// TIA Portal V17 export
// export: Created 2023-09-14T22:30:54.9161637Z, ExportSetting WithDefaults, DisplayName Totally Integrated Automation Portal, DisplayVersion V17 Update 6, DisplayName TIA Portal Openness, DisplayVersion V17 Update 6, DisplayName TIA Portal Teamcenter Gateway, DisplayVersion V17 Update 6, DisplayName TIA Portal Version Control Interface, DisplayVersion V17, DisplayName Simotion SCOUT TIA, DisplayVersion 5.4.3.0, DisplayName TIA Portal Test Suite Advanced, DisplayVersion V17 Update 1, DisplayName SIMOCODE ES, DisplayVersion V17 Update 5, DisplayName SINAMICS Startdrive Advanced, DisplayVersion V17 SP1, DisplayName SINAMICS Startdrive G130, G150, S120, S150, SINAMICS MV, S210, DisplayVersion V17 SP1, DisplayName SINAMICS Startdrive G110M, G120, G120C, G120D, G120P, G115D, DisplayVersion V17 SP1, DisplayName SIRIUS Safety ES, DisplayVersion V17 Update 5, DisplayName STEP 7 Professional, DisplayVersion V17 Update 6, DisplayName STEP 7 CFC, DisplayVersion V17 Update 1, DisplayName STEP 7 Safety, DisplayVersion V17 Update 6, DisplayName WinCC Advanced, DisplayVersion V17 Update 6, DisplayName SIMATIC Visualization Architect, DisplayVersion V17 Update 5
DATA_BLOCK "08_AL_FILTER"   // DB26
{ S7_Optimized_Access := 'TRUE' }
VERSION : 0.1
// stored: AutoNumber true, DBAccessibleFromOPCUA true, DBAccessibleFromWebserver true, IsOnlyStoredInLoadMemory false, IsRetainMemResEnabled false, IsWriteProtectedInAS false, MemoryReserve 100
   VAR
      "n0006-zp001-el001-k25501_SN50" : Bool;
      "n0007-zp001-el001-k25502_SN50" : Bool;
      "n0008-zp001-el001-k25601_SN50" : Bool;
      "n0009-zp001-el001-k25602_SN50" : Bool;
      "n0005-zp001-el001-k40001_SN50" : Bool;
      "n0013-uf317-xn10_SN50" : Bool;
      "n0015-uc16-el001-k30001_SN50" : Bool;
      "n0016-uc164-xn10_SN50" : Bool;
      "n0017-lv004-el001-k30001_SN50" : Bool;
      "n0018-lv004-el001-k30001_SN50" : Bool;
      "n0020-uc15-el001-k30001_SN50" : Bool;
      "n0023-uc154-xn10_SN50" : Bool;
      "n0021-icg11-el001-k30001_SN50" : Bool;
      "n0022-icg21-el001-k30001_SN50" : Bool;
      "n0025-uc14-el001-k30001_SN50" : Bool;
      "n0026-uc144-xn10_SN50" : Bool;
      "n0038-uc1-el001-k30001_SN50" : Bool;
      "n0039-lv001-el001-k30001_SN50" : Bool;
      "n0040-lv001-el001-k30001_SN50" : Bool;
      "n0041-uf31-el002-k30001_SN50" : Bool;
      "n0042-uf41-el002-k30001_SN50" : Bool;
      "n0044-ct1-el001-k30001_SN50" : Bool;
      "n0045-ct1-el002-k30001_SN50" : Bool;
      "n0046-ct1-el003-k30001_SN50" : Bool;
      "n0047-lv002-el001-k30001_SN50" : Bool;
      "n0048-lv002-el001-k30001_SN50" : Bool;
      "n0050-uc13-el001-k30001_SN50" : Bool;
      "n0051-uc134-xn10_SN50" : Bool;
      "n0053-uc12-el001-k30001_SN50" : Bool;
      "n0055-uc124-xn10_SN50" : Bool;
      "n0054-uf31-el003-k30001_SN50" : Bool;
      "n0057-uc11-el001-k30001_SN50" : Bool;
      "n0060-uc114-xn10_SN50" : Bool;
      "n0058-lv003-el001-k30001_SN50" : Bool;
      "n0059-lv003-el001-k30001_SN50" : Bool;
      "n0028-uc17-el001-k30001_SN50" : Bool;
      "n0029-uc173-xn10_SN50" : Bool;
      "n0010-zp001-el001-k24501_SN50" : Bool;
      "n0033-zp001-el001-k40001_SN50" : Bool;
      "n0034-ug6-el001-k30001_SN50" : Bool;
      "n0035-ug6-xn10_SN50" : Bool;
      "n0043-db93-el001-k30001_SN50" : Bool;
      "n0031-db931-xn10_SN50" : Bool;
      "n0005-lv008-el001-k30001_SN51" : Bool;
      "n0006-lv008-el001-k30001_SN51" : Bool;
      "n0007-icg22-el001-k30001_SN51" : Bool;
      "n0008-icg12-el001-k30001_SN51" : Bool;
      "n0009-uf42-el002-k30001_SN51" : Bool;
      "n0010-lv007-el001-k30001_SN51" : Bool;
      "n0011-lv007-el001-k30001_SN51" : Bool;
      "n0021-uc2-el001-k30001_SN51" : Bool;
      "n0025-dc91-el001-k30001_SN51" : Bool;
      "n0026-uc915-xn10_SN51" : Bool;
      "n0027-uc915-xn11_SN51" : Bool;
      "n0028-lv005-el001-k30001_SN51" : Bool;
      "n0029-ct2-el001-k30001_SN51" : Bool;
      "n0033-uc26-el001-k30001_SN51" : Bool;
      "n0034-uc264-xn10_SN51" : Bool;
      "n0035-ct2-el002-k30001_SN51" : Bool;
      "n0036-lv005-el001-k30001_SN51" : Bool;
      "n0041-uc27-el001-k30001_SN51" : Bool;
      "n0042-uc274-xn10_SN51" : Bool;
      "n0046-uc25-el001-k30001_SN51" : Bool;
      "n0047-uc254-xn10_SN51" : Bool;
      "n0048-lv006-el001-k30001_SN51" : Bool;
      "n0051-uc24-el001-k30001_SN51" : Bool;
      "n0052-uc244-xn10_SN51" : Bool;
      "n0056-uc23-el001-k30001_SN51" : Bool;
      "n0057-uc234-xn10_SN51" : Bool;
      "n0058-ct2-el003-k30001_SN51" : Bool;
      "n0061-uc22-el001-k30001_SN51" : Bool;
      "n0062-uc224-xn10_SN51" : Bool;
      "n0063-lv006-el001-k30001_SN51" : Bool;
      "n0066-uc21-el001-k30001_SN51" : Bool;
      "n0067-uc214-xn10_SN51" : Bool;
      "n0070-uf31-el001-k30001_SN51" : Bool;
      "n0071-uf41-el001-k30001_SN51" : Bool;
      "n0072-uf51-el001-k30001_SN51" : Bool;
      "n0080-uf511-xn10_SN51" : Bool;
      "n0073-ifg31-el001-k30001_SN51" : Bool;
      "n0074-ifg41-el001-k30001_SN51" : Bool;
      "n0075-uf32-el001-k30001_SN51" : Bool;
      "n0076-uf42-el001-k30001_SN51" : Bool;
      "n0082-zp002-el001-k30001_SN51" : Bool;
      "n0083-lv001-el001-k30001_SN51" : Bool;
      "n0084-lv001-el001-k30001_SN51" : Bool;
      "n0085-uc29-el001-k30001_SN51" : Bool;
      "n0092-zp001-el001-k24501_SN51" : Bool;
      "n0091-zp001-el001-k30001_SN51" : Bool;
      "n0093-ug7-el001-k30001_SN51" : Bool;
      "n0094-ug7-xn10_SN51" : Bool;
   END_VAR
BEGIN
END_DATA_BLOCK
